FUNCTION_BLOCK TONReset EXTENDS TON
VAR_INPUT
END_VAR
VAR_OUTPUT
	rtTimerDone	: R_TRIG;
END_VAR
VAR
END_VAR

SUPER^();

rtTimerDone(CLK	:= THIS^.Q);

IF THIS^.Q THEN 
	THIS^.IN	:= FALSE;
END_IF

END_FUNCTION_BLOCK

(* stored: Version 1.1.0.1, ProductVersion 3.1.4024.9
   POU TONReset: Id {68f1984f-e7b4-4af0-ba3c-91ded775ff11}, SpecialFunc None *)
